// TIA Portal V15 export
// export: Created 2019-05-03T16:21:01.4579834Z, ExportSetting WithDefaults, DisplayName Totally Integrated Automation Portal, DisplayVersion V15, DisplayName TIA Portal Openness, DisplayVersion V15, DisplayName STEP 7 Professional, DisplayVersion V15, DisplayName STEP 7 Safety, DisplayVersion V15, DisplayName WinCC Professional, DisplayVersion V15, DisplayName SIMATIC Visualization Architect, DisplayVersion V15
VAR_GLOBAL   // PLC tag table "ROBNAME"
END_VAR
